FUNCTION_BLOCK CylControlChan (* Composite Function Block Type *)
  (* Standard: 61499-2 *)
  (* Version 0.0, 7/14/2023, valeriy, nxtControl GmBH, template *)
  PACKAGE Main;
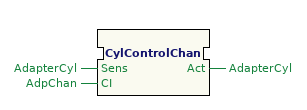
  SOCKETS
    Sens : AdapterCyl;
    CI : AdpChan;
  END_SOCKETS
  PLUGS
    Act : AdapterCyl;
  END_PLUGS
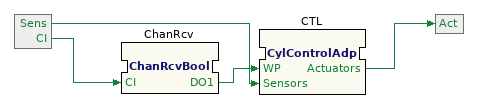
  FBS
    ChanRcv : ChanRcvBool;
    CTL : CylControlAdp;
  END_FBS
  ADAPTER_CONNECTIONS
    ChanRcv.DO1 TO CTL.WP;
    CI TO ChanRcv.CI;
    CTL.Actuators TO Act;
    Sens TO CTL.Sensors;
  END_CONNECTIONS
END_FUNCTION_BLOCK
